FUNCTION FC_ProductStatus : eProductStatus
VAR_INPUT
	aByte					: stByteAsBit;
END_VAR

IF aByte.aBit.b0 THEN
	IF aByte.aBit.b1 THEN
		FC_ProductStatus := eProductStatus.Scraped;
	ELSIF aByte.aBit.b3 THEN
		FC_ProductStatus := eProductStatus.Completed;
	ELSIF aByte.aBit.b2 THEN
		FC_ProductStatus := eProductStatus.Working;	
	ELSE
		FC_ProductStatus := eProductStatus.Present;
	END_IF
ELSE
	FC_ProductStatus := eProductStatus.NotPresent;
END_IF

END_FUNCTION

(* stored: Version 1.1.0.1, ProductVersion 3.1.4024.15
   POU FC_ProductStatus: Id {5e0bec4e-aa0b-473e-b9b1-6db8b30792e7}, SpecialFunc None *)
